FUNCTION_BLOCK FB_MotionAxisNC_Test EXTENDS FB_TestSuite
VAR
    fbHome : FB_HomeNC_TestDouble;
    fbHalt : FB_HaltNC_TestDouble;
    fbPower : FB_PowerNC_TestDouble;
    fbReset : FB_ResetNC_TestDouble;
    fbMoveAbsolute : FB_MoveAbsoluteNC_TestDouble;
    fbReadParameter : FB_ReadParameterNC_TestDouble;
    fbWriteParameter  : FB_WriteParameterNC_TestDouble;
    fbParamSaveRestore: FB_ParamSaveRestoreNC_TestDouble;
    fbEncoderScaling : FB_EncoderScalingNC_TestDouble;
    fbAxisStatus : FB_AxisStatusNC_TestDouble;
    fbBacklashCompensation : FB_BacklashCompensationNC_TestDouble;

END_VAR

GivenAllMCBlockErrorConditionThenPowerErrorHasHigherPriority();

METHOD PRIVATE GivenAllMCBlockErrorConditionThenPowerErrorHasHigherPriority
VAR_INST
    // subject under test
    fbMotionAxis : FB_MotionAxisNC(  	iHome := fbHome,
                                        iHalt := fbHalt,
                                        iPower := fbPower,
                                        iReset := fbReset,
                                        iMoveAbsolute := fbMoveAbsolute,
                                        iReadParameter := fbReadParameter,
                                        iWriteParameter  := fbWriteParameter,
                                        iParamSaveRestore:= fbParamSaveRestore,
                                        iEncoderScaling := fbEncoderScaling,
                                        iAxisStatus := fbAxisStatus,
                                        iBacklashCompensation := fbBacklashCompensation
                                    );
bExpectedAxisError :BOOL := TRUE;
nExpectedErrorId: UDINT;
END_VAR
TEST(__POUNAME());

    // Power highest priority
    fbHome.Error := TRUE;
    fbHalt.Error := TRUE;
    fbPower.Error := TRUE;
    fbReset.Error := TRUE;
    fbMoveAbsolute.Error := TRUE;
    fbReadParameter.Error := TRUE;
    fbWriteParameter.Error := TRUE;
    fbParamSaveRestore.Error := TRUE;
    fbAxisStatus.Error := TRUE;
    fbBacklashCompensation.Error := TRUE;
    fbMotionAxis();

    nExpectedErrorId := 18000;
    AssertTrue(Condition :=  fbMotionAxis.Status.bError, Message := 'Prioritized and generalized Error must be set #1');
    AssertEquals_UDINT ( Expected:=nExpectedErrorId , Actual:=fbMotionAxis.Status.nErrorID, Message:='Prioritized error Id must be 18000 #2');

    // Halt has 2nd highest priority
    fbHome.Error := TRUE;
    fbHalt.Error := TRUE;
    fbPower.Error := FALSE;
    fbReset.Error := TRUE;
    fbMoveAbsolute.Error := TRUE;
    fbReadParameter.Error := TRUE;
    fbWriteParameter.Error := TRUE;
    fbParamSaveRestore.Error := TRUE;
    fbAxisStatus.Error := TRUE;
    fbBacklashCompensation.Error := TRUE;
    fbMotionAxis();

    nExpectedErrorId := 19000;
    AssertTrue(Condition :=  fbMotionAxis.Status.bError, Message := 'Prioritized and generalized Error must be set #3');
    AssertEquals_UDINT ( Expected:=nExpectedErrorId , Actual:=fbMotionAxis.Status.nErrorID, Message:='Prioritized error Id must be 19000 #4');

    // Reset 3rd highest priority
    fbHome.Error := TRUE;
    fbHalt.Error := FALSE;
    fbPower.Error := FALSE;
    fbReset.Error := TRUE;
    fbMoveAbsolute.Error := TRUE;
    fbReadParameter.Error := TRUE;
    fbWriteParameter.Error := TRUE;
    fbParamSaveRestore.Error := TRUE;
    fbAxisStatus.Error := TRUE;
    fbBacklashCompensation.Error := TRUE;
    fbMotionAxis();

    nExpectedErrorId := 20000;
    AssertTrue(Condition :=  fbMotionAxis.Status.bError, Message := 'Prioritized and generalized Error must be set #5');
    AssertEquals_UDINT ( Expected:=nExpectedErrorId , Actual:=fbMotionAxis.Status.nErrorID, Message:='Prioritized error Id must be 20000 #6');

    // BacklashCompensation 4th highest priority
    fbHome.Error := TRUE;
    fbHalt.Error := FALSE;
    fbPower.Error := FALSE;
    fbReset.Error := FALSE;
    fbMoveAbsolute.Error := TRUE;
    fbReadParameter.Error := TRUE;
    fbWriteParameter.Error := TRUE;
    fbParamSaveRestore.Error := TRUE;
    fbAxisStatus.Error := TRUE;
    fbBacklashCompensation.Error := TRUE;
    fbMotionAxis();

    nExpectedErrorId := 21000;
    AssertTrue(Condition :=  fbMotionAxis.Status.bError, Message := 'Prioritized and generalized Error must be set #7');
    AssertEquals_UDINT ( Expected:=nExpectedErrorId , Actual:=fbMotionAxis.Status.nErrorID, Message:='Prioritized error Id must be 21000 #8');

    // MoveAbsolute 5th highest priority
    fbHome.Error := TRUE;
    fbHalt.Error := FALSE;
    fbPower.Error := FALSE;
    fbReset.Error := FALSE;
    fbMoveAbsolute.Error := TRUE;
    fbReadParameter.Error := TRUE;
    fbWriteParameter.Error := TRUE;
    fbParamSaveRestore.Error := TRUE;
    fbAxisStatus.Error := TRUE;
    fbBacklashCompensation.Error := FALSE;
    fbMotionAxis();

    nExpectedErrorId := 22000;
    AssertTrue(Condition :=  fbMotionAxis.Status.bError, Message := 'Prioritized and generalized Error must be set #9');
    AssertEquals_UDINT ( Expected:=nExpectedErrorId , Actual:=fbMotionAxis.Status.nErrorID, Message:='Prioritized error Id must be 22000 #10');

    // Home 6th highest priority
    fbHome.Error := TRUE;
    fbHalt.Error := FALSE;
    fbPower.Error := FALSE;
    fbReset.Error := FALSE;
    fbMoveAbsolute.Error := FALSE;
    fbReadParameter.Error := TRUE;
    fbWriteParameter.Error := TRUE;
    fbParamSaveRestore.Error := TRUE;
    fbAxisStatus.Error := TRUE;
    fbBacklashCompensation.Error := FALSE;
    fbMotionAxis();

    nExpectedErrorId := 23000;
    AssertTrue(Condition :=  fbMotionAxis.Status.bError, Message := 'Prioritized and generalized Error must be set #11');
    AssertEquals_UDINT ( Expected:=nExpectedErrorId , Actual:=fbMotionAxis.Status.nErrorID, Message:='Prioritized error Id must be 23000 #12');

    // AxisError 7th highest priority
    fbHome.Error := FALSE;
    fbHalt.Error := FALSE;
    fbPower.Error := FALSE;
    fbReset.Error := FALSE;
    fbMoveAbsolute.Error := FALSE;
    fbReadParameter.Error := TRUE;
    fbWriteParameter.Error := TRUE;
    fbParamSaveRestore.Error := TRUE;
    fbAxisStatus.Error := TRUE;
    fbBacklashCompensation.Error := FALSE;
    fbMotionAxis();

    nExpectedErrorId := 24000;
    AssertTrue(Condition :=  fbMotionAxis.Status.bError, Message := 'Prioritized and generalized Error must be set #13');
    AssertEquals_UDINT ( Expected:=nExpectedErrorId , Actual:=fbMotionAxis.Status.nErrorID, Message:='Prioritized error Id must be 24000 #14');

    // ReadParameters 8th highest priority
    fbHome.Error := FALSE;
    fbHalt.Error := FALSE;
    fbPower.Error := FALSE;
    fbReset.Error := FALSE;
    fbMoveAbsolute.Error := FALSE;
    fbReadParameter.Error := TRUE;
    fbWriteParameter.Error := TRUE;
    fbParamSaveRestore.Error := TRUE;
    fbAxisStatus.Error := FALSE;
    fbBacklashCompensation.Error := FALSE;
    fbMotionAxis();

    nExpectedErrorId := 25000;
    AssertTrue(Condition :=  fbMotionAxis.Status.bError, Message := 'Prioritized and generalized Error must be set #15');
    AssertEquals_UDINT ( Expected:=nExpectedErrorId , Actual:=fbMotionAxis.Status.nErrorID, Message:='Prioritized error Id must be 25000 #16');

    // WriteParameters 8th highest priority
    fbHome.Error := FALSE;
    fbHalt.Error := FALSE;
    fbPower.Error := FALSE;
    fbReset.Error := FALSE;
    fbMoveAbsolute.Error := FALSE;
    fbReadParameter.Error := FALSE;
    fbWriteParameter.Error := TRUE;
    fbParamSaveRestore.Error := TRUE;
    fbAxisStatus.Error := FALSE;
    fbBacklashCompensation.Error := FALSE;
    fbMotionAxis();

    nExpectedErrorId := 26000;
    AssertTrue(Condition :=  fbMotionAxis.Status.bError, Message := 'Prioritized and generalized Error must be set #17');
    AssertEquals_UDINT ( Expected:=nExpectedErrorId , Actual:=fbMotionAxis.Status.nErrorID, Message:='Prioritized error Id must be 26000 #18');

    // save Restore 9th highest priority
    fbHome.Error := FALSE;
    fbHalt.Error := FALSE;
    fbPower.Error := FALSE;
    fbReset.Error := FALSE;
    fbMoveAbsolute.Error := FALSE;
    fbReadParameter.Error := FALSE;
    fbWriteParameter.Error := FALSE;
    fbParamSaveRestore.Error := TRUE;
    fbAxisStatus.Error := FALSE;
    fbBacklashCompensation.Error := FALSE;
    fbMotionAxis();

    nExpectedErrorId := 27000;
    AssertTrue(Condition :=  fbMotionAxis.Status.bError, Message := 'Prioritized and generalized Error must be set #19');
    AssertEquals_UDINT ( Expected:=nExpectedErrorId , Actual:=fbMotionAxis.Status.nErrorID, Message:='Prioritized error Id must be 27000 #20');

TEST_FINISHED();
END_METHOD

END_FUNCTION_BLOCK

(* stored: Version 1.1.0.1
   POU FB_MotionAxisNC_Test: Id {fa75d716-c423-459e-9a73-6d09eee7d5ba}, SpecialFunc None
   Method GivenAllMCBlockErrorConditionThenPowerErrorHasHigherPriority: Id {9c82fcc9-f025-46d3-bdb0-63a901189948} *)
